// TIA Portal V19 export
// export: Created 2026-08-09T01:52:25.0422155Z, ExportSetting WithDefaults, DisplayName Totally Integrated Automation Portal, DisplayVersion V19, DisplayName TIA Portal Openness, DisplayVersion V19, DisplayName TIA Portal Version Control Interface, DisplayVersion V19, DisplayName STEP 7 Professional, DisplayVersion V19, DisplayName STEP 7 Safety, DisplayVersion V19, DisplayName WinCC Basic/Comfort/Advanced, DisplayVersion V19, DisplayName WinCC Unified, DisplayVersion V19
DATA_BLOCK "dc_DB"   // DB4
VERSION : 0.1
// stored: AutoNumber true, DBAccessibleFromOPCUA true, DBAccessibleFromWebserver true, InstanceOfName dc, InstanceOfType FB
"dc"
   // VAR_INPUT
   //    timePt : Time;
   // END_VAR
   // VAR_OUTPUT
   //    timeQ : Bool;
   // END_VAR
   // VAR
   //    timeP : Bool;
   //    timeS : Bool;
   // END_VAR
BEGIN
END_DATA_BLOCK
